TEXTLIST EspesorTabla
  0 = 'Sin seleccionar'
  1 = '3'
  2 = '6'
  3 = '12'
  4 = '20'
   = ''
END_TEXTLIST

(* stored: Version 1.1.0.1, ProductVersion 3.1.4024.12
   TextList EspesorTabla: Id {22e4705c-dacd-4e35-9954-cfc1d2caef47} *)
